// Update the height of material in the tank
FUNCTION UpdateHigh

VAR
	// Flow in [m3/s]
	in : REAL := GVL.flow_in; // m3/s
	
	// Flow out [m3/s]
	out : REAL := FlowOut(); // m3/s
	
	// Coeff
	coef : REAL := GVL.time_step / GVL.tank_area; // s/m2
	
	// delta
	dhigh : REAL; // m3/s * s/m2 -> m
	
END_VAR

dhigh := (in - out) * coef;
GVL.high_now := GVL.high_now + dhigh;

GVL.volPC_now := GVL.high_now * 100 / GVL.tank_high;

END_FUNCTION

(* stored: Version 1.1.0.1, ProductVersion 3.1.4024.12
   POU UpdateHigh: Id {ddacef68-b9e7-4d3b-a171-9a0343e6bd9b}, SpecialFunc None *)
